{attribute 'qualified_only'}
{attribute 'strict'}
{attribute 'to_string'}
TYPE E_AxisHomingDirection :
(
    None     := 0,//无方向
    Positive := 10,//正向
    Negative := 20//负向
);
END_TYPE

(* stored: Version 1.1.0.1, ProductVersion 3.1.4026.20
   DUT E_AxisHomingDirection: Id {65e70f71-6a68-4b54-b767-acde68823465} *)
